// TIA Portal V17 export
// export: Created 2025-05-06T14:29:00.6601383Z, ExportSetting WithDefaults, DisplayName Totally Integrated Automation Portal, DisplayVersion V17 Update 8, DisplayName TIA Portal Openness, DisplayVersion V17 Update 8, DisplayName TIA Portal Version Control Interface, DisplayVersion V17, DisplayName SINAMICS Startdrive Advanced, DisplayVersion V17 SP2, DisplayName SINAMICS Startdrive G110M, G120, G120C, G120D, G120P, G115D, DisplayVersion V17 SP2, DisplayName SINAMICS Startdrive G130, G150, S120, S150, SINAMICS MV, S210, DisplayVersion V17 SP2, DisplayName STEP 7 Professional, DisplayVersion V17 Update 8, DisplayName SINUMERIK ONE STEP 7 Toolbox, DisplayVersion V17 Update 12, DisplayName SINUMERIK 840D sl STEP 7 Toolbox, DisplayVersion V17 Update 12, DisplayName STEP 7 Safety, DisplayVersion V17 Update 6, DisplayName WinCC Advanced, DisplayVersion V17 Update 8
DATA_BLOCK "DB7270_HMI_LUBRICATION_CONTROL"   // DB7270
{ S7_Optimized_Access := 'FALSE' }
AUTHOR : ETXETAR
VERSION : 1.0
// stored: AutoNumber false, DBAccessibleFromOPCUA true, DBAccessibleFromWebserver true, IsOnlyStoredInLoadMemory false, IsWriteProtectedInAS false
   VAR RETAIN
      CAPTURE_DATA : Struct
         LUBRICATION_CYCLE_START : Bool;   // LUBRICATION CYCLE START
         LUBRICATION_CYCLE_FINISH : Bool;   // LUBRICATION CYCLE FINISH
         LUBR_CAPTURE_DATA_START : Bool;   // LUBRICATION CAPTURE DATA START
         LUBRICATION_DONE_OK : Bool;   // LUBRICATION DONE OK
         LUBRICATION_DONE_NOK : Bool;   // LUBRICATION DONE NOK
         LUBRICATION_P_PULSE : Bool;   // LUBRICATION POSITIVE PULSE
         LUBRICATION_N_PULSE : Bool;   // LUBRICATION NEGATIVE PULSE
         ACTUAL_LUBRIC_DATE : Date;   // ACTUAL LUBRICATION DATE
         ACTUAL_LUBRIC_START_TIME : Time_Of_Day;   // ACTUAL LUBRICATION START TIME
         ACTUAL_LUBRIC_FINISH_TIME : Time_Of_Day;   // ACTUAL LUBRICATION FINISH TIME
      END_STRUCT;
      VISU_HMI_DATE : Struct
         LAST_LUBRIC_DATE_1 : Date;   // LAST LUBRICATION DATE 1
         LAST_LUBRIC_DATE_2 : Date;   // LAST LUBRICATION DATE 2
         LAST_LUBRIC_DATE_3 : Date;   // LAST LUBRICATION DATE 3
         LAST_LUBRIC_DATE_4 : Date;   // LAST LUBRICATION DATE 4
         LAST_LUBRIC_DATE_5 : Date;   // LAST LUBRICATION DATE 5
         LAST_LUBRIC_DATE_6 : Date;   // LAST LUBRICATION DATE 6
         LAST_LUBRIC_DATE_7 : Date;   // LAST LUBRICATION DATE 7
         LAST_LUBRIC_DATE_8 : Date;   // LAST LUBRICATION DATE 8
         LAST_LUBRIC_DATE_9 : Date;   // LAST LUBRICATION DATE 9
         LAST_LUBRIC_DATE_10 : Date;   // LAST LUBRICATION DATE 10
      END_STRUCT;
      VISU_HMI_TIME_START : Struct
         LAST_LUBRIC_START_TIME_1 : Time_Of_Day;   // LAST LUBRICATION START TIME 1
         LAST_LUBRIC_START_TIME_2 : Time_Of_Day;   // LAST LUBRICATION START TIME 2
         LAST_LUBRIC_START_TIME_3 : Time_Of_Day;   // LAST LUBRICATION START TIME 3
         LAST_LUBRIC_START_TIME_4 : Time_Of_Day;   // LAST LUBRICATION START TIME 4
         LAST_LUBRIC_START_TIME_5 : Time_Of_Day;   // LAST LUBRICATION START TIME 5
         LAST_LUBRIC_START_TIME_6 : Time_Of_Day;   // LAST LUBRICATION START TIME 6
         LAST_LUBRIC_START_TIME_7 : Time_Of_Day;   // LAST LUBRICATION START TIME 7
         LAST_LUBRIC_START_TIME_8 : Time_Of_Day;   // LAST LUBRICATION START TIME 8
         LAST_LUBRIC_START_TIME_9 : Time_Of_Day;   // LAST LUBRICATION START TIME 9
         LAST_LUBRIC_START_TIME_10 : Time_Of_Day;   // LAST LUBRICATION START TIME 10
      END_STRUCT;
      VISU_HMI_TIME_FINISH : Struct
         LAST_LUBRIC_FINISH_TIME_1 : Time_Of_Day;   // LAST LUBRICATION FINISH TIME 1
         LAST_LUBRIC_FINISH_TIME_2 : Time_Of_Day;   // LAST LUBRICATION FINISH TIME 2
         LAST_LUBRIC_FINISH_TIME_3 : Time_Of_Day;   // LAST LUBRICATION FINISH TIME 3
         LAST_LUBRIC_FINISH_TIME_4 : Time_Of_Day;   // LAST LUBRICATION FINISH TIME 4
         LAST_LUBRIC_FINISH_TIME_5 : Time_Of_Day;   // LAST LUBRICATION FINISH TIME 5
         LAST_LUBRIC_FINISH_TIME_6 : Time_Of_Day;   // LAST LUBRICATION FINISH TIME 6
         LAST_LUBRIC_FINISH_TIME_7 : Time_Of_Day;   // LAST LUBRICATION FINISH TIME 7
         LAST_LUBRIC_FINISH_TIME_8 : Time_Of_Day;   // LAST LUBRICATION FINISH TIME 8
         LAST_LUBRIC_FINISH_TIME_9 : Time_Of_Day;   // LAST LUBRICATION FINISH TIME 9
         LAST_LUBRIC_FINISH_TIME_10 : Time_Of_Day;   // LAST LUBRICATION FINISH TIME 10
      END_STRUCT;
      VISU_HMI_DONE : Struct
         LUBRI_STATUS_DONE_1 : Bool;   // LUBRICATION STATUS DONE 1
         LUBRI_STATUS_DONE_2 : Bool;   // LUBRICATION STATUS DONE 2
         LUBRI_STATUS_DONE_3 : Bool;   // LUBRICATION STATUS DONE 3
         LUBRI_STATUS_DONE_4 : Bool;   // LUBRICATION STATUS DONE 4
         LUBRI_STATUS_DONE_5 : Bool;   // LUBRICATION STATUS DONE 5
         LUBRI_STATUS_DONE_6 : Bool;   // LUBRICATION STATUS DONE 6
         LUBRI_STATUS_DONE_7 : Bool;   // LUBRICATION STATUS DONE 7
         LUBRI_STATUS_DONE_8 : Bool;   // LUBRICATION STATUS DONE 8
         LUBRI_STATUS_DONE_9 : Bool;   // LUBRICATION STATUS DONE 9
         LUBRI_STATUS_DONE_10 : Bool;   // LUBRICATION STATUS DONE 10
      END_STRUCT;
      REQUEST_LUBRICATION_BY_DAYS : Bool;   // REQUEST LUBRICATION BY DAYS
      ACTUAL_DATE : Date;   // ACTUAL DATE
   END_VAR
BEGIN
END_DATA_BLOCK
